FUNCTION_BLOCK FB_StringLookupLREALMock EXTENDS FB_FalliblePublicMock IMPLEMENTS I_StringLookupLREAL
VAR
    fValue : LREAL;
END_VAR


METHOD Lookup : LREAL
VAR_INPUT
    StringToLookup	: T_MaxString;
END_VAR

Lookup := fValue;
END_METHOD


METHOD SetValid

ClearError();
END_METHOD

PROPERTY Value : LREAL
GET

Value := fValue;
END_GET
SET

fValue := Value;
END_SET
END_PROPERTY

END_FUNCTION_BLOCK

(* stored: Version 1.1.0.1
   POU FB_StringLookupLREALMock: Id {682595e9-23e7-433f-b4e7-703251f5a029}, SpecialFunc None
   Method Lookup: Id {630af135-431d-4e29-ba31-858823424239}
   Method SetValid: Id {d166fb74-2990-4b60-a23f-5d3fe53ca986}
   Property Value: Id {1a2296e6-151f-4fc5-818d-1a3ab6f535e7}
   Get Get: Id {0676378a-fc9d-475f-9e99-03547d0a3663}
   Set Set: Id {6b9486c5-a536-4abc-befd-6b1a14c80d31} *)
